RoboDK station: pizza_order_demo.rdk

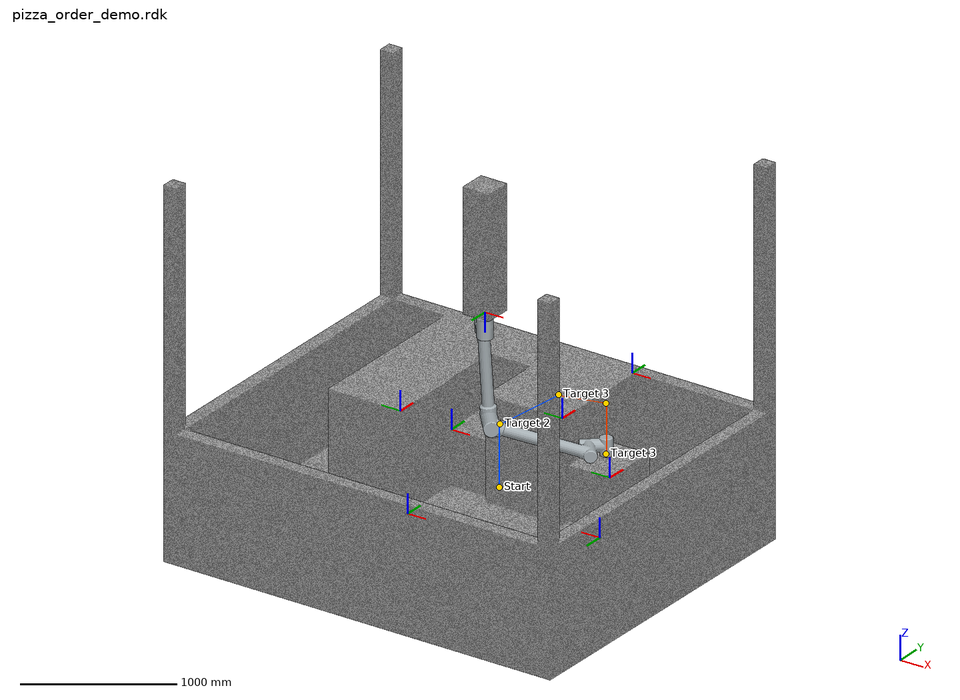
[picture v0: the station drawn from its stored meshes, robots at their saved joint values, targets as dots, program paths as lines]
Station pizza_order_demo (saved by RoboDK 5.4.0). Poses are relative to the parent item; angles as X-Y-Z fixed-axis rotations.
  - frame Avena arm Base at (607.5, -10, 1600) mm, rotated rx 180 ry 0 rz 0 deg
    - robot Avena arm: 6 axes
        modified DH rows (alpha deg, a mm, theta deg, d mm): 0, 0, 0, 123.3; 90, 0, 90, 0; 0, 686, 0, 0; 0, 671, -90, 116.4; -90, 0, 0, 115.4; 90, 0, 0, 67.4
        joint limits [-174.7, -90, -166, -174.7, -174.7, -174.7] to [174.7, 90, 166, 174.7, 174.7, 174.7]; home [0, 0, 0, 0, 0, 0]; saved at [-40.64, -3.293, -67.167, -19.541, -90, -49.36]
  - object kontener v08 stp at (0, 0, 0) mm, size 3000 x 2500 x 2665 mm, geometry from kontener v08 stp.stp
  - frame Oven entry at (1229, 491, 400) mm, rotated rx 0 ry 0 rz 90 deg
  - frame Oven exit at (0, 491, 400) mm
  - frame Conveyor at (0, -80, 760) mm, rotated rx 0 ry 0 rz 90 deg
  - frame Display at (909.02, 420, 760) mm, rotated rx 0 ry 0 rz 90 deg
  - frame Storage base at (1215, 400, 10) mm, rotated rx 0 ry 0 rz 180 deg
  - Python program Visualize Trajectory (listed below)
  - frame Pick piece from display at (0, 0, 0) mm
    - target Start (Cartesian target) at (752.42, -54.52, 418.54) mm, rotated rx -180 ry 0 rz 90 deg; joints [67.232, 43.561, -86.194, -47.367, -90, -67.232] of Avena arm
    - target Target 2 (Cartesian target) at (756.99, -56.66, 866.55) mm, rotated rx 180 ry 0 rz 180 deg; joints [65.346, 66.099, -132.855, -23.245, -90, -155.346] of Avena arm
    - target Target 3 (Cartesian target) at (809.02, 520, 860) mm, rotated rx 180 ry 0 rz 180 deg; joints [-57.336, 19.068, -117.557, 8.49, -90, -32.664] of Avena arm
  - frame Place piece in oven at (0, 2491, 0) mm
    - target Target 1 (Cartesian target) at (809.02, -1971, 860) mm, rotated rx 180 ry 0 rz 180 deg; joints [-57.336, 19.068, -117.557, 8.49, -90, -32.664] of Avena arm
    - target Target 2 (Cartesian target) at (1129, -1900, 860) mm, rotated rx 180 ry 0 rz 180 deg; joints [-40.64, -1.236, -100.505, 11.741, -90, -49.36] of Avena arm
    - target Target 3 (Cartesian target) at (1129, -1900, 500) mm, rotated rx 180 ry 0 rz 180 deg; joints [-40.64, -3.293, -67.167, -19.541, -90, -49.36] of Avena arm
  - program PickPieceFromDisplay (4 instructions, listed below)
  - program PlacePieceInOven (4 instructions, listed below)
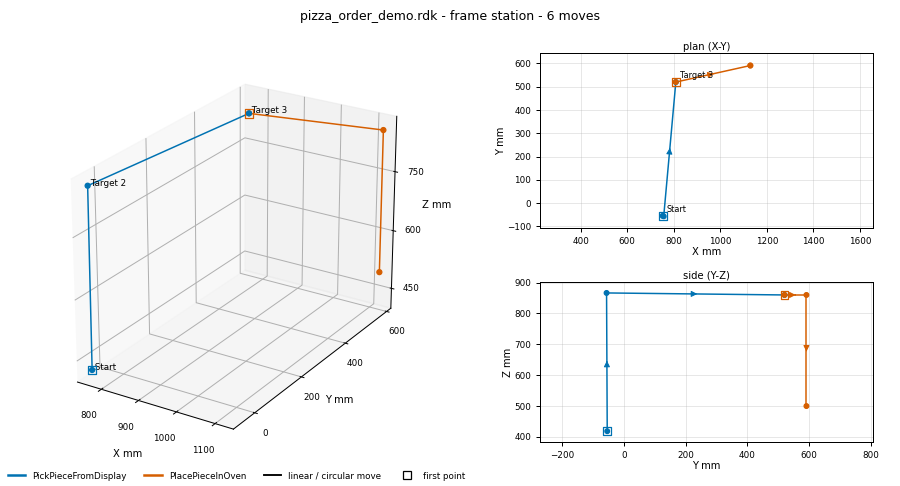
[picture p0: tool path of pizza_order_demo.rdk in frame station, 6 of 6 moves have a stored position in this frame; points joined in program order, loops and branches not executed]

--- Python program Visualize Trajectory ---
# Type help("robodk.robolink") or help("robodk.robomath") for more information
# Press F5 to run the script
# Documentation: https://robodk.com/doc/en/RoboDK-API.html
# Reference:     https://robodk.com/doc/en/PythonAPI/index.html
# Note: It is not required to keep a copy of this file, your Python script is saved with your RDK project
import time
from robodk import robolink, robomath, robodialogs

# if __name__ == '__main__':
RDK = robolink.Robolink()

progname = robodialogs.mbox("Name of program: ", entry='Prog1')

program = RDK.Item(progname)
if not program.Valid():
    RDK.ShowMessage(f'There is no program with name "{progname}"')
else:
    message, traj, status = program.InstructionListJoints(flags=4, time_step=0.01)
    if status < 0:
        RDK.ShowMessage(f'Failed to generate valid trajectory.\nMessage: {message}\nStatus: {status}')
        exit(1)

    traj = traj.list2()
    if len(traj) < 2:
        RDK.ShowMessage('Cannot replay robot path because number of trajectory points is too low.')
        exit(1)
    else:
        robot = RDK.Item('Avena arm')
        for jtp in traj:
            joint_angles, time_step = jtp[:6], jtp[10]
            robot.setJoints(joint_angles)
            time.sleep(time_step)

--- program PickPieceFromDisplay (robot Avena arm) ---
  Set Ref.: Pick piece from display
  MoveJ (Start)
  MoveL (Target 2)
  MoveL (Target 3)

--- program PlacePieceInOven (robot Avena arm) ---
  Set Ref.: Place piece in oven
  MoveJ (Target 1)
  MoveL (Target 2)
  MoveL (Target 3)
